PROGRAM P_Demo_PDINT_TO_DINT
VAR
    nRealValue           : DINT := -123456; // 模拟 wire 缓冲区中的 DINT 字段
    pDINTField           : POINTER TO DINT; // 业务侧先算好的字段地址（ADR 或 pBase+nOff）
    bExtractField        : BOOL; // 在线置 TRUE 触发一次解析
    nRealValue_extracted : DINT; // 解析后的副本，供业务逻辑使用
END_VAR

// ============================================================
// Tc2_Utilities.PDINT_TO_DINT 演示程序（FUNCTION）
// ============================================================
// 场景：从一段二进制 wire 缓冲区里按偏移取 DINT 字段（Modbus/CAN/ADS Raw）。
// 价值：替代手写 pField + nOff + ^ 指针算术；一次调用取值，少打错符号。
// 验证：在线写 nRealValue := -123456；bExtractField := TRUE；
//       下一周期 nRealValue_extracted 应等于 nRealValue。
// ============================================================

// 业务代码通常已经算好字段地址（pBase + 协议偏移）；演示用 ADR 等价
pDINTField := ADR(nRealValue);

IF bExtractField AND pDINTField <> 0 THEN
    // 单次完整调用：避免手写 ^ 解引用，统一风格便于和字节序转换串联
    nRealValue_extracted := PDINT_TO_DINT(pDINTField);
    bExtractField := FALSE;
END_IF;

END_PROGRAM

(* stored: Version 1.1.0.1, ProductVersion 3.1.4024.5
   POU P_Demo_PDINT_TO_DINT: Id {27d160d0-f36a-5017-8910-44617f3c2fe9}, SpecialFunc None *)
